// TIA Portal V18 export
TYPE "PartDataHMI"
   STRUCT
      PartQuality : DInt;   // 当前物料的剩余数量 / Remaining quantity of current material
      BoxDisplayID { S7_SetPoint := 'True'} : Int;   // 显示料盒编号 / Display material box number
      PartQualitySet : DInt;   // 当前物料的剩余数量 / Remaining quantity of current material
      CMD : Struct   // 人工设定数量值 / Manually set quantity value
         ClearCurrentBox : Bool;
         ClearAllBox : Bool;
         "PartQuality+1" : Bool;
         "PartQuality-1" : Bool;
         PartQualityAck : Bool;   // 人工输入值确认 / Manually input value confirmation
      END_STRUCT;
      Waring : Struct
         Insufficient : Bool;   // 物料不足，请扫码添加 / Insufficient material, please scan to add
         BufferBoxFull : Bool;   // 物料缓存已满，无法添加 / Material cache full, unable to add
         ScannCodeInvalid : Bool;   // 扫的物料码无效，或已经已用过 / Invalid material code scanned, or already used
      END_STRUCT;
      PartDataDispaly : "PartCodeStruct_UDT";
   END_STRUCT;
END_TYPE
